// TIA Portal V17 export
// export: Created 2024-09-02T12:50:33.3494294Z, ExportSetting WithDefaults, DisplayName Totally Integrated Automation Portal, DisplayVersion V17, DisplayName TIA Portal Openness, DisplayVersion V17, DisplayName TIA Portal Version Control Interface, DisplayVersion V17, DisplayName STEP 7 Professional, DisplayVersion V17, DisplayName STEP 7 Safety, DisplayVersion V17, DisplayName WinCC Professional, DisplayVersion V17
TYPE "TypeMobySequenzBIS"
// stored: IsFailsafeCompliant false
   STRUCT
      AuftFach : Struct   // Auftragsfach / Job mailbox
         SequenzNr : Int;   // aktuelle Sequenznummer / current sequence number
         Funktion : Int;   // 1= Lesen; 2= Schreiben / 1= Read; 2= Write
         ADDR_TAG : DInt;   // Adresse auf dem MDS / Address on the MDS
         LEN_DATA : DInt;   // Anzahl Byte für Auftrag / Number of bytes for job
      END_STRUCT;
      ErgFach : Struct   // Ergebnisfach / Result compartment
         SequenzNr : Int;   // aktuelle Sequenznummer / current sequence number
         Funktion : Int;   // 1= Lesen; 2= Schreiben / 1= Read; 2= Write
         BereitFürAuftrag : Bool;   // ASM Bereit für Auftrag / ASM Ready for order
      END_STRUCT;
   END_STRUCT;
END_TYPE
